FUNCTION_BLOCK TEST_NEN (* Test NE functions of numerical values *)
  (* Standard: IEC 61499-1 *)
  (* Version 0.0, 2006-09-11, JHC, Holobloc Inc *)
  (* Compiler header: package fb.rt.test; *)
  (* Compiler classdef: SimpleFB *)
  (* Compiler Java Sun JDK 1.5.0 *)
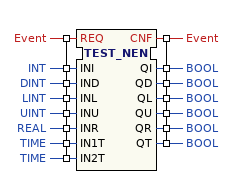
  EVENT_INPUT
    REQ WITH INI, INL, INU, IND, INR, IN1T, IN2T;
  END_EVENT
  EVENT_OUTPUT
    CNF WITH QI, QD, QL, QU, QR, QT;
  END_EVENT
  VAR_INPUT
    INI : INT;
    IND : DINT;
    INL : LINT;
    INU : UINT;
    INR : REAL;
    IN1T : TIME;
    IN2T : TIME;
  END_VAR
  VAR_OUTPUT
    QI : BOOL;
    QD : BOOL;
    QL : BOOL;
    QU : BOOL;
    QR : BOOL;
    QT : BOOL;
  END_VAR
  ALGORITHM REQ IN FBD:
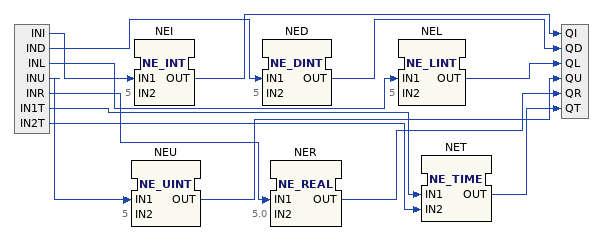
    FBS
      NEI : NE_INT(IN2 := 5);
      NED : NE_DINT(IN2 := 5);
      NEL : NE_LINT(IN2 := 5);
      NEU : NE_UINT(IN2 := 5);
      NER : NE_REAL(IN2 := 5.0);
      NET : NE_TIME;
    END_FBS
    DATA_CONNECTIONS
      INI TO NEI.IN1;
      IND TO NED.IN1;
      INL TO NEL.IN1;
      INU TO NEU.IN1;
      INR TO NER.IN1;
      NEI.OUT TO QI;
      NED.OUT TO QD;
      NEL.OUT TO QL;
      NEU.OUT TO QU;
      NER.OUT TO QR;
      NET.OUT TO QT;
      IN1T TO NET.IN1;
      IN2T TO NET.IN2;
    END_CONNECTIONS
  END_ALGORITHM
END_FUNCTION_BLOCK
